{attribute 'qualified_only'}
{attribute 'strict'}
TYPE E_SpeedControlState :
(
	STOPPED,
	ACCELERATE,
	RUNNING,
	DECELERATE
);
END_TYPE

(* stored: Version 1.1.0.1, ProductVersion 3.1.4022.12
   DUT E_SpeedControlState: Id {144af7ab-b13e-4b60-8aef-b0e46a69915a} *)
